// TIA Portal V17 export
// export: Created 2024-08-09T12:53:13.9426664Z, ExportSetting WithDefaults, DisplayName Totally Integrated Automation Portal, DisplayVersion V17 Update 7, DisplayName TIA Portal Openness, DisplayVersion V17 Update 7, DisplayName TIA Portal Version Control Interface, DisplayVersion V17, DisplayName STEP 7 Professional, DisplayVersion V17 Update 7, DisplayName STEP 7 Safety, DisplayVersion V17 Update 6, DisplayName WinCC Professional, DisplayVersion V17 Update 7
VAR_GLOBAL   // PLC tag table "MELANGEUSE"
END_VAR
VAR_GLOBAL CONSTANT   // user constants
   NIV_MLG_DEBUT_LOT : USInt := 1;
   NIV_MLG_PRETE : USInt := 5;
   NIV_MLG_MARCHE : USInt := 10;
   NIV_MLG_DEBUT_REMP : USInt := 15;
   NIV_MLG_FIN_REMP : USInt := 20;
   NIV_MLG_FIN_PREMELANG : USInt := 30;
   NIV_MLG_FIN_INJ_LIQ : USInt := 40;
   NIV_MLG_PRESQ_FINI : USInt := 50;
   NIV_MLG_PRETE_VIDANGE : USInt := 70;
   NIV_MLG_OUVERTE : USInt := 80;
   NIV_MLG_DEBUT_TEMPO_VIDANGE : USInt := 90;
   NIV_MLG_FIN_LOT : USInt := 255;
END_VAR
